TYPE LG_Coils :
STRUCT
	b_EnableOperation			:	BOOL := FALSE;
	b_EnableSwwOperation		: 	BOOL := FALSE;
	b_EnableSilentMode			:	BOOL := FALSE;
	b_EnableDesinfectionMode	:	BOOL := FALSE;
	b_EmstopActive				:	BOOL := FALSE;
	b_EnableEmStop				:	BOOL := FALSE;
END_STRUCT
END_TYPE

(* stored: Version 1.1.0.1, ProductVersion 3.1.4026.18
   DUT LG_Coils: Id {2cf45aff-0d37-48e8-a1fc-d67235f6996c} *)
